FUNCTION "Main stazioni" : Void
{ S7_Optimized_Access := 'TRUE' }
VERSION : 0.1
   VAR_TEMP
      CounterStazioni : Int;
      CounterDestinazioni : Int;
      K_Analogica : Int;
      DisabilitaStazioneAdditiva : Bool;
      CondizioniTimeout : Bool;
   END_VAR


BEGIN
	IF "Stazione".Funzioni.Inizializza THEN
	    FOR #CounterStazioni := 0 TO "K_NumStazione" DO
	        FOR #CounterDestinazioni := 0 TO "K_NumStazione" DO
	            "Stazione".S[#CounterStazioni].Destinazione[#CounterDestinazioni].IN.Possibile := False;
	        END_FOR;
	        "Stazione".S[#CounterStazioni].Hmi.Diagnostica.TroppoPieno :=
	        "Stazione".S[#CounterStazioni].Dati.InvioAdditivo.Abilitazione :=
	        "Stazione".S[#CounterStazioni].Dati.InvioAdditivo.Attiva :=
	        "Stazione".S[#CounterStazioni].Dati.RicezioneAdditivo.Attiva :=
	        "Stazione".S[#CounterStazioni].Dati.GestionePrioritàAttiva.DaDestinazione :=
	        "Stazione".S[#CounterStazioni].Dati.GestionePrioritàAttiva.DaSorgente :=
	        "Stazione".S[#CounterStazioni].Dati.AlmenoUnaDestinazioneProgettata :=
	        "Stazione".S[#CounterStazioni].Dati.AlmenoUnaSorgenteProgettata :=
	        "Stazione".S[#CounterStazioni].Prm.AbilitazionePriorità.SuEstrazioni :=
	        "Stazione".S[#CounterStazioni].Prm.AbilitazionePriorità.SugliArrivi :=
	        "Stazione".S[#CounterStazioni].Prm.IgnoraDestinazione :=
	        "Stazione".S[#CounterStazioni].Prm.ByPassChiamataDestinazione := False;
	        "Stazione".S[#CounterStazioni].Dati.K_StazioneDestinazione :=
	        "Stazione".S[#CounterStazioni].Dati.InvioAdditivo.K_StazioneMandata1 :=
	        "Stazione".S[#CounterStazioni].Dati.RicezioneAdditivo.K_StazioneAdditivo1 := 0;
	        "Stazione".S[#CounterStazioni].IN.SorgenteNonPronta :=
	        "Stazione".S[#CounterStazioni].IN.LivelloDestinazioneSuperiorePriorità :=
	        "Stazione".S[#CounterStazioni].IN.LivelloSorgenteInferiorePriorità := False;
	    END_FOR;
	    "Stazione".Hmi.AggiornaConfigurazione := True;
	    "Stazione".Funzioni.Inizializza := False;
	END_IF;
END_FUNCTION

